Staubli VAL3: ReplyCode.pjx

--- ReplyCode.pjx ---
Parameters version=s7.8.1 stackSize=5000 millimeterUnit=true
Program file=start.pgx
Program file=stop.pgx
Data file=ReplyCode.dtx

--- ReplyCode.dtx ---
public num INVALID
public num SUCCESS
public num FAILURE
